// This interface provides a method to retrieve descriptive messages for error codes.
INTERFACE I_ErrorDescriptor EXTENDS __SYSTEM.IQueryInterface;

// Retrieves the descriptive message for the specified error code.
METHOD GetDescription : T_ErrorMessage // The descriptive message corresponding to the provided error code.
VAR_INPUT
	Code : T_ErrorCode; // The error code for which the description is to be retrieved.
END_VAR
END_METHOD

END_INTERFACE

(* stored: Version 1.1.0.1
   Itf I_ErrorDescriptor: Id {1e09aa87-89c5-07d8-3cda-a921df257785}
   Method GetDescription: Id {a1f7ef42-61c8-068c-1500-e81800f8675c} *)
